// TIA Portal V16 export
// export: Created 2022-07-21T09:35:31.0085271Z, ExportSetting WithDefaults, DisplayName Totally Integrated Automation Portal, DisplayVersion V16 Update 4, DisplayName TIA Portal Version Control Interface, DisplayVersion V16 Update 2, DisplayName TIA Portal Openness, DisplayVersion V16 Update 4, DisplayName SINAMICS Startdrive Advanced, DisplayVersion V16 Update 5, DisplayName SINAMICS Startdrive G130, G150, S120, S150, SINAMICS MV, S210, DisplayVersion V16 Update 5, DisplayName SINAMICS Startdrive G110M, G120, G120C, G120D, G120P, G115D, DisplayVersion V16 Update 5, DisplayName STEP 7 Professional, DisplayVersion V16 Update 4, DisplayName STEP 7 Safety, DisplayVersion V16, DisplayName WinCC Advanced, DisplayVersion V16 Update 4
FUNCTION_BLOCK "fbPhotocell"   // FB32, LAD
TITLE = Photocell handling / Obsługa fotoceli
{ S7_Optimized_Access := 'TRUE' }
VERSION : 0.1
// stored: AutoNumber true, IsIECCheckEnabled false, IsRetainMemResEnabled false, MemoryReserve 100, SetENOAutomatically false, UDAEnableTagReadback false
   VAR_INPUT
      inEnable { ExternalAccessible := 'False'; ExternalVisible := 'False'; ExternalWritable := 'False'} : Bool;   // Zezwolenie ogólne / General release
      inPhotocellNC { ExternalAccessible := 'False'; ExternalVisible := 'False'; ExternalWritable := 'False'} : Bool;   // Wejście z fotokomórki / Photocell input
      inResetFault { ExternalAccessible := 'False'; ExternalVisible := 'False'; ExternalWritable := 'False'} : Bool;   // Reset błędu / Error reset
      inAutomatic { ExternalAccessible := 'False'; ExternalVisible := 'False'; ExternalWritable := 'False'} : Bool;   // Tryb automatyczny / Automatic mode
      inDistancePrevScan { ExternalAccessible := 'False'; ExternalVisible := 'False'; ExternalWritable := 'False'} : USInt;   // Dystans / Distance
      inDistanceShifting : UInt;   // Przesunięcie wirtualne fotoceli / Virtual photocell shift
      inClearMessageCounter { ExternalAccessible := 'False'; ExternalVisible := 'False'; ExternalWritable := 'False'} : Bool;   // Wyczyszczenie pamięci licznika okupacji / Clear occupation counter
      inAllowResetIfOccupied { ExternalAccessible := 'False'; ExternalVisible := 'False'; ExternalWritable := 'False'} : Bool;   // Pozwolenie na reset błędu fotoceli, gdy jest zajęta / Permission to reset photocell error, when occupied
      inFilterPecOccupied { ExternalAccessible := 'False'; ExternalVisible := 'False'; ExternalWritable := 'False'} : UInt;   // Filtrowanie sygnały okupacji fotoceli / Occupation signal filter
      inFilterPecFree { ExternalAccessible := 'False'; ExternalVisible := 'False'; ExternalWritable := 'False'} : UInt;   // Filtrowanie zejścia sygnału okupacji fotoceli / No occupation signal filter
      inDistanceUntilMessage { ExternalAccessible := 'False'; ExternalVisible := 'False'; ExternalWritable := 'False'} : UInt := 0;   // Dystans, po którym pojawi się błąd / Distance to error
   END_VAR
   VAR_OUTPUT
      ouFeedbackPhotocell { ExternalAccessible := 'False'; ExternalVisible := 'False'; ExternalWritable := 'False'} : "typePhotocell";   // Struktura fotoceli / Photocell structure
      ouPhotocellBlocked { ExternalAccessible := 'False'; ExternalVisible := 'False'; ExternalWritable := 'False'} : Bool;   // Błąd, fotocela zablokowana / Error, photocell locked
      ouCommand : "typeCommand";   // Komenda sygnałowa / Signal command
   END_VAR
   VAR
      sPositiveEdge { ExternalAccessible := 'False'; ExternalVisible := 'False'; ExternalWritable := 'False'} : Bool;
      snegativeEdge { ExternalAccessible := 'False'; ExternalVisible := 'False'; ExternalWritable := 'False'} : Bool;
      sEdgeAutomatic { ExternalAccessible := 'False'; ExternalVisible := 'False'; ExternalWritable := 'False'} : Bool;
      sCounterDebounceFree { ExternalAccessible := 'False'; ExternalVisible := 'False'; ExternalWritable := 'False'} : UInt;
      sCounterDebounceOccupied { ExternalAccessible := 'False'; ExternalVisible := 'False'; ExternalWritable := 'False'} : UInt;
      sCounterMessageBlocked { ExternalAccessible := 'False'; ExternalVisible := 'False'; ExternalWritable := 'False'} : UInt;
      sMonitoringBlocked { S7_SetPoint := 'True'} : "fbError";
      sShiftSignal { S7_SetPoint := 'True'} : "fbShifting";
      sBufferArray { S7_SetPoint := 'True'} : Array[0..30] of "typeSignalBuffer";
   END_VAR
   VAR_TEMP
      tEdgeAutomatic : Bool;
      tReleaseCounter : Bool;
      tResetEnergySaving : Bool;
      tResetBlocked : Bool;
      tInternalEnable : Bool;
   END_VAR
   VAR_TEMP   // added for the SCL form of the ladder/FBD networks
      _w1 : Bool;
   END_VAR
BEGIN

REGION Network 1: Temporary variables / Wypracowanie zmiennych tymczasowych
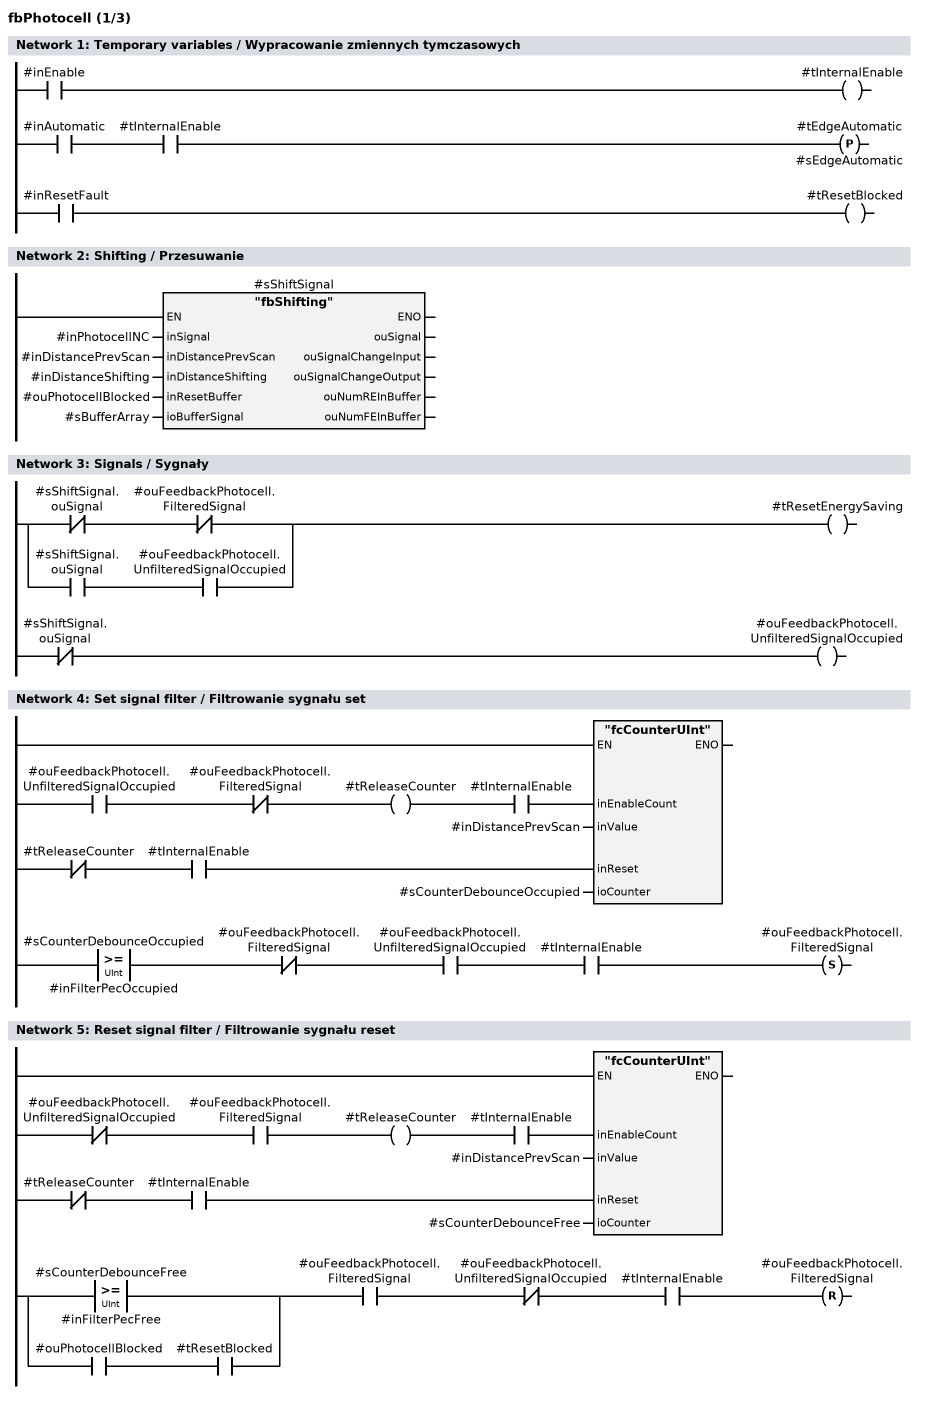
   #tInternalEnable := #inEnable;
   #_w1 := #inAutomatic AND #tInternalEnable;
   #tEdgeAutomatic := #_w1 AND NOT #sEdgeAutomatic;   // rising edge
   #sEdgeAutomatic := #_w1;
   #tResetBlocked := #inResetFault;
END_REGION

REGION Network 2: Shifting / Przesuwanie
   RUNG wire#powerrail
      #sShiftSignal(inSignal := #inPhotocellNC, inDistancePrevScan := #inDistancePrevScan, inDistanceShifting := #inDistanceShifting, inResetBuffer := #ouPhotocellBlocked, ioBufferSignal := #sBufferArray, ouSignal =>, ouSignalChangeInput =>, ouSignalChangeOutput =>, ouNumREInBuffer =>, ouNumFEInBuffer =>)
   END_RUNG
   // the same network as SCL:
   #sShiftSignal(inSignal := #inPhotocellNC,   // "fbShifting"
                 inDistancePrevScan := #inDistancePrevScan,
                 inDistanceShifting := #inDistanceShifting,
                 inResetBuffer := #ouPhotocellBlocked,
                 ioBufferSignal := #sBufferArray);
END_REGION

REGION Network 3: Signals / Sygnały
   RUNG wire#powerrail
      I_Contact( #sShiftSignal.ouSignal )
      I_Contact( #ouFeedbackPhotocell.FilteredSignal )
      wire#w1
      Coil( #tResetEnergySaving )
   END_RUNG
   RUNG wire#powerrail
      Contact( #sShiftSignal.ouSignal )
      Contact( #ouFeedbackPhotocell.UnfilteredSignalOccupied )
   END_RUNG wire#w1
   RUNG wire#powerrail
      I_Contact( #sShiftSignal.ouSignal )
      Coil( #ouFeedbackPhotocell.UnfilteredSignalOccupied )
   END_RUNG
   // the same network as SCL:
   #tResetEnergySaving := (NOT #sShiftSignal.ouSignal AND NOT #ouFeedbackPhotocell.FilteredSignal) OR (#sShiftSignal.ouSignal AND #ouFeedbackPhotocell.UnfilteredSignalOccupied);
   #ouFeedbackPhotocell.UnfilteredSignalOccupied := NOT #sShiftSignal.ouSignal;
END_REGION

REGION Network 4: Set signal filter / Filtrowanie sygnału set
   RUNG wire#powerrail
      "fcCounterUInt"(inEnableCount := wire#w1, inReset := wire#w2, inValue := #inDistancePrevScan, ioCounter := #sCounterDebounceOccupied)
   END_RUNG
   RUNG wire#powerrail
      Contact( #ouFeedbackPhotocell.UnfilteredSignalOccupied )
      I_Contact( #ouFeedbackPhotocell.FilteredSignal )
      Coil( #tReleaseCounter )
      Contact( #tInternalEnable )
   END_RUNG wire#w1
   RUNG wire#powerrail
      I_Contact( #tReleaseCounter )
      Contact( #tInternalEnable )
   END_RUNG wire#w2
   RUNG wire#powerrail
      { S7_Templates := "SrcType := UInt" } GE_Contact(in1 := #sCounterDebounceOccupied, in2 := #inFilterPecOccupied)
      I_Contact( #ouFeedbackPhotocell.FilteredSignal )
      Contact( #ouFeedbackPhotocell.UnfilteredSignalOccupied )
      Contact( #tInternalEnable )
      S_Coil( #ouFeedbackPhotocell.FilteredSignal )
   END_RUNG
   // the same network as SCL:
   #tReleaseCounter := #ouFeedbackPhotocell.UnfilteredSignalOccupied AND NOT #ouFeedbackPhotocell.FilteredSignal;
   "fcCounterUInt"(inEnableCount := #tReleaseCounter AND #tInternalEnable,
                   inValue := #inDistancePrevScan,
                   inReset := NOT #tReleaseCounter AND #tInternalEnable,
                   ioCounter := #sCounterDebounceOccupied);
   IF (#sCounterDebounceOccupied >= #inFilterPecOccupied) AND NOT #ouFeedbackPhotocell.FilteredSignal AND #ouFeedbackPhotocell.UnfilteredSignalOccupied AND #tInternalEnable THEN
       #ouFeedbackPhotocell.FilteredSignal := TRUE;
   END_IF;
END_REGION

REGION Network 5: Reset signal filter / Filtrowanie sygnału reset
   RUNG wire#powerrail
      "fcCounterUInt"(inEnableCount := wire#w1, inReset := wire#w2, inValue := #inDistancePrevScan, ioCounter := #sCounterDebounceFree)
   END_RUNG
   RUNG wire#powerrail
      I_Contact( #ouFeedbackPhotocell.UnfilteredSignalOccupied )
      Contact( #ouFeedbackPhotocell.FilteredSignal )
      Coil( #tReleaseCounter )
      Contact( #tInternalEnable )
   END_RUNG wire#w1
   RUNG wire#powerrail
      I_Contact( #tReleaseCounter )
      Contact( #tInternalEnable )
   END_RUNG wire#w2
   RUNG wire#powerrail
      { S7_Templates := "SrcType := UInt" } GE_Contact(in1 := #sCounterDebounceFree, in2 := #inFilterPecFree)
      wire#w3
      Contact( #ouFeedbackPhotocell.FilteredSignal )
      I_Contact( #ouFeedbackPhotocell.UnfilteredSignalOccupied )
      Contact( #tInternalEnable )
      R_Coil( #ouFeedbackPhotocell.FilteredSignal )
   END_RUNG
   RUNG wire#powerrail
      Contact( #ouPhotocellBlocked )
      Contact( #tResetBlocked )
   END_RUNG wire#w3
   // the same network as SCL:
   #tReleaseCounter := NOT #ouFeedbackPhotocell.UnfilteredSignalOccupied AND #ouFeedbackPhotocell.FilteredSignal;
   "fcCounterUInt"(inEnableCount := #tReleaseCounter AND #tInternalEnable,
                   inValue := #inDistancePrevScan,
                   inReset := NOT #tReleaseCounter AND #tInternalEnable,
                   ioCounter := #sCounterDebounceFree);
   IF ((#sCounterDebounceFree >= #inFilterPecFree) OR (#ouPhotocellBlocked AND #tResetBlocked)) AND #ouFeedbackPhotocell.FilteredSignal AND NOT #ouFeedbackPhotocell.UnfilteredSignalOccupied AND #tInternalEnable THEN
       #ouFeedbackPhotocell.FilteredSignal := FALSE;
   END_IF;
END_REGION

REGION Network 6: Occupation / Zajętość
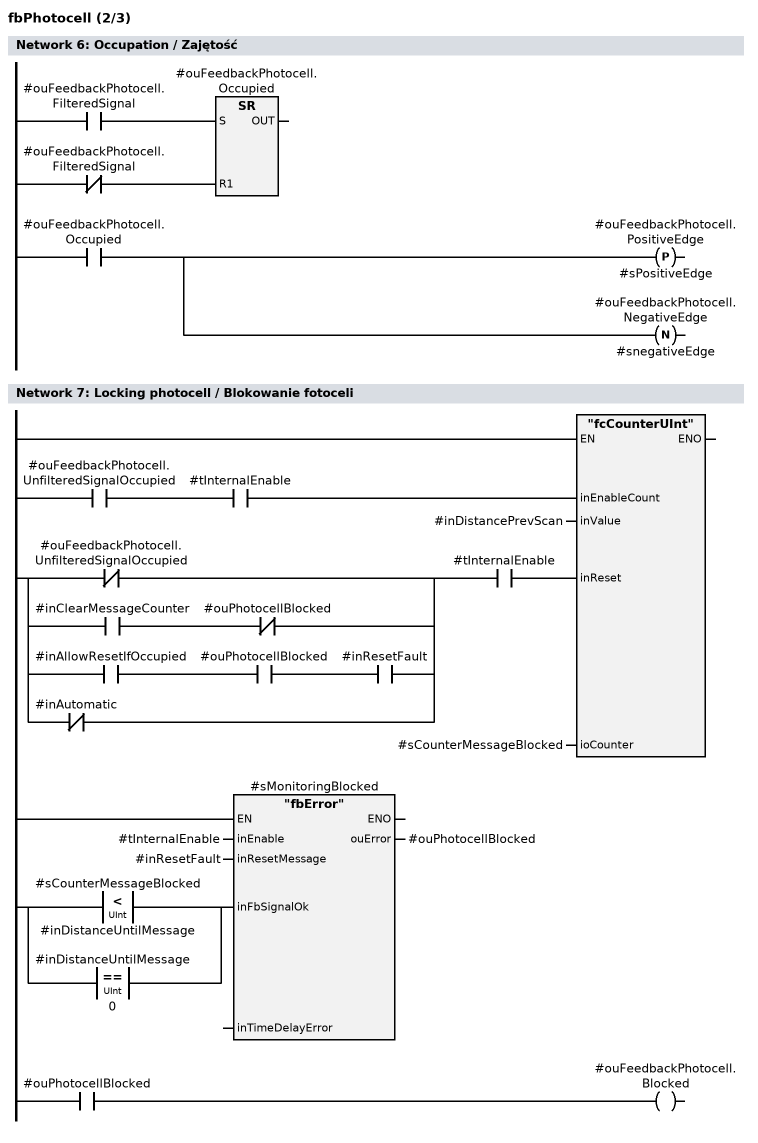
   IF #ouFeedbackPhotocell.FilteredSignal THEN
       #ouFeedbackPhotocell.Occupied := TRUE;   // SR flip-flop
   END_IF;
   IF NOT #ouFeedbackPhotocell.FilteredSignal THEN #ouFeedbackPhotocell.Occupied := FALSE; END_IF;
   #ouFeedbackPhotocell.PositiveEdge := #ouFeedbackPhotocell.Occupied AND NOT #sPositiveEdge;   // rising edge
   #sPositiveEdge := #ouFeedbackPhotocell.Occupied;
   #ouFeedbackPhotocell.NegativeEdge := NOT #ouFeedbackPhotocell.Occupied AND #snegativeEdge;   // falling edge
   #snegativeEdge := #ouFeedbackPhotocell.Occupied;
END_REGION

REGION Network 7: Locking photocell / Blokowanie fotoceli
   RUNG wire#powerrail
      "fcCounterUInt"(inEnableCount := wire#w1, inReset := wire#w3, inValue := #inDistancePrevScan, ioCounter := #sCounterMessageBlocked)
   END_RUNG
   RUNG wire#powerrail
      Contact( #ouFeedbackPhotocell.UnfilteredSignalOccupied )
      Contact( #tInternalEnable )
   END_RUNG wire#w1
   RUNG wire#powerrail
      I_Contact( #ouFeedbackPhotocell.UnfilteredSignalOccupied )
      wire#w2
      Contact( #tInternalEnable )
   END_RUNG wire#w3
   RUNG wire#powerrail
      Contact( #inClearMessageCounter )
      I_Contact( #ouPhotocellBlocked )
   END_RUNG wire#w2
   RUNG wire#powerrail
      Contact( #inAllowResetIfOccupied )
      Contact( #ouPhotocellBlocked )
      Contact( #inResetFault )
   END_RUNG wire#w2
   RUNG wire#powerrail
      I_Contact( #inAutomatic )
   END_RUNG wire#w2
   RUNG wire#powerrail
      #sMonitoringBlocked(inFbSignalOk := wire#w4, inEnable := #tInternalEnable, inResetMessage := #inResetFault, inTimeDelayError :=, ouError => #ouPhotocellBlocked)
   END_RUNG
   RUNG wire#powerrail
      { S7_Templates := "SrcType := UInt" } LT_Contact(in1 := #sCounterMessageBlocked, in2 := #inDistanceUntilMessage)
   END_RUNG wire#w4
   RUNG wire#powerrail
      { S7_Templates := "SrcType := UInt" } EQ_Contact(in1 := #inDistanceUntilMessage, in2 := 0)
   END_RUNG wire#w4
   RUNG wire#powerrail
      Contact( #ouPhotocellBlocked )
      Coil( #ouFeedbackPhotocell.Blocked )
   END_RUNG
   // the same network as SCL:
   "fcCounterUInt"(inEnableCount := #ouFeedbackPhotocell.UnfilteredSignalOccupied AND #tInternalEnable,
                   inValue := #inDistancePrevScan,
                   inReset := (NOT #ouFeedbackPhotocell.UnfilteredSignalOccupied OR (#inClearMessageCounter AND NOT #ouPhotocellBlocked) OR (#inAllowResetIfOccupied AND #ouPhotocellBlocked AND #inResetFault) OR NOT #inAutomatic) AND #tInternalEnable,
                   ioCounter := #sCounterMessageBlocked);
   #sMonitoringBlocked(inEnable := #tInternalEnable,   // "fbError"
                       inResetMessage := #inResetFault,
                       inFbSignalOk := (#sCounterMessageBlocked < #inDistanceUntilMessage) OR (#inDistanceUntilMessage = 0),
                       ouError => #ouPhotocellBlocked);
   #ouFeedbackPhotocell.Blocked := #ouPhotocellBlocked;
END_REGION

REGION Network 8: Signal command / Komenda sygnałowa
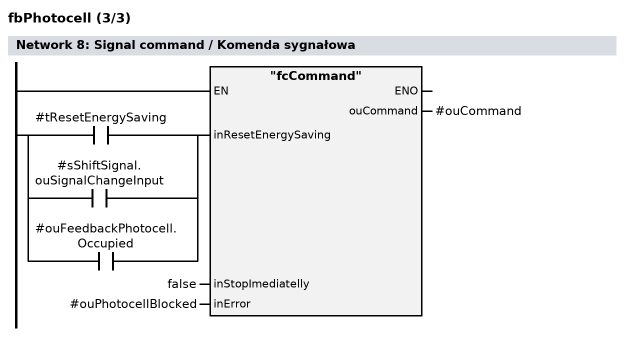
   RUNG wire#powerrail
      "fcCommand"(inResetEnergySaving := wire#w1, inStopImediatelly := false, inError := #ouPhotocellBlocked, ouCommand => #ouCommand)
   END_RUNG
   RUNG wire#powerrail
      Contact( #tResetEnergySaving )
   END_RUNG wire#w1
   RUNG wire#powerrail
      Contact( #sShiftSignal.ouSignalChangeInput )
   END_RUNG wire#w1
   RUNG wire#powerrail
      Contact( #ouFeedbackPhotocell.Occupied )
   END_RUNG wire#w1
   // the same network as SCL:
   "fcCommand"(inResetEnergySaving := #tResetEnergySaving OR #sShiftSignal.ouSignalChangeInput OR #ouFeedbackPhotocell.Occupied,
               inStopImediatelly := false,
               inError := #ouPhotocellBlocked,
               ouCommand => #ouCommand);
END_REGION
END_FUNCTION_BLOCK
